// TwinCAT 3 PLC project ccslib
// Title: ESO ELT CCS Library
// Company: ESO
// Author: Mario Kiekebusch
// ProjectVersion: 0.0.1.0
// Description: ELT - CCS Library providing FB helping to receive deterministic data via MUDPI.
// ProgramVersion: 3.1.4022.4
// libraries:
//   ESO ELT Utility Library, * (ESO)
//   ESO LDC Common Library, * (ESO)
//   ESO LDC Timer Library, * (ESO)
//   ESO MUDPI Library, * (ESO)
//   Tc2_EtherCAT, * (Beckhoff Automation GmbH)
//   Tc2_Standard, * (Beckhoff Automation GmbH)
//   Tc2_System, * (Beckhoff Automation GmbH)
//   Tc2_Utilities, * (Beckhoff Automation GmbH)
//   Tc3_Module, * (Beckhoff Automation GmbH)
//   VisuDialogs, * (System)
//   VisuSymbols,3.5.10.0,System
// project tree:
//   DUTs/Structures/ T_CCS_GUI.TcDUT, T_DATA_SAMPLE.TcDUT
//   / GlobalTextList.TcGTLO, VisualizationManager.TcVMO (not stored)
//   GVLs/ GCL.TcGVL, GVL_TimeConstants.TcGVL
//   POUs/ FB_CCS_RECEIVER.TcPOU, FB_LINEAR_INTERPOLATION.TcPOU, MAIN.TcPOU
//   Version/ Global_Version.TcGVL
//   VISUs/Templates/ GUI_TEMPLATE_CCS_RECEIVER.TcVIS

// ---- DUTs/Structures/T_CCS_GUI.TcDUT
TYPE T_CCS_GUI :
STRUCT
	alt: LREAL;
	az: LREAL;
	pa: LREAL;
	time_tai: STRING;
	lst: LREAL;
	ra: LREAL;
	dec: LREAL;
	north_angle: LREAL;
	pupil_angle: LREAL;
	ha: LREAL;
END_STRUCT
END_TYPE

// ---- DUTs/Structures/T_DATA_SAMPLE.TcDUT
TYPE T_DATA_SAMPLE :
STRUCT
	value: LREAL := 0.0;
	timestamp: LREAL := 0.0;
END_STRUCT
END_TYPE

// ---- GVLs/GCL.TcGVL
{attribute 'qualified_only'}
VAR_GLOBAL
	C_PI:				LREAL := 3.1415926535897932384626433832795028841971693993751;
    C_PI2: 				LREAL := C_PI / 2.0;
	C_2PI: 				LREAL := 2.0 * C_PI;
END_VAR

// ---- GVLs/GVL_TimeConstants.TcGVL
{attribute 'qualified_only'}
VAR_GLOBAL
	C_INVALID:    DINT := -9999;
	C_ONE_SEC:    LINT := 1000000000;
	C_STAT_OK:    DINT := 0;
	C_NS2MSEC:    LREAL := 1/1E+6;
	C_NS2SEC:     LREAL := 1/1E+9;
	C_UNIX_OFFSET_SEC: ULINT := DATE_TO_ULINT(DATE#2000-01-01); // 946,684,800 seconds = 15,778,080 minutes = 262,968 hours
	C_UNIX_OFFSET_MICROSEC:  ULINT := C_UNIX_OFFSET_SEC * 10#1000_000;
END_VAR

// ---- Version/Global_Version.TcGVL
{attribute 'TcGenerated'}
{attribute 'no-analysis'}
{attribute 'linkalways'}
// This function has been automatically generated from the project information.
VAR_GLOBAL CONSTANT
	{attribute 'const_non_replaced'}
	stLibVersion_ESO_ELT_CCS_Library : ST_LibVersion := (iMajor := 0, iMinor := 0, iBuild := 1, iRevision := 0, nFlags := 0, sVersion := '0.0.1.0');
END_VAR

// ---- POUs/FB_CCS_RECEIVER.TcPOU
FUNCTION_BLOCK FB_CCS_RECEIVER
VAR_INPUT
	refTimeObj  : REFERENCE TO FB_TIME; 
END_VAR
VAR_OUTPUT
END_VAR
VAR
	fbMudpiReceiver: FB_MUDPI_RECEIVER;
	tracking_raw : T_ASTRO_POINTING_KERNEL_POSITIONS;
	tracking_ccs : T_CCS_GUI;
	north_sample: T_DATA_SAMPLE;
	pupil_sample: T_DATA_SAMPLE;
	pa_sample: T_DATA_SAMPLE;
	north_angle_interpolator: FB_LINEAR_INTERPOLATION;
	pupil_angle_interpolator: FB_LINEAR_INTERPOLATION;
	pa_angle_interpolator: FB_LINEAR_INTERPOLATION;
	previous_sample_id: UDINT := 0;
	
	
  
	
	
END_VAR

// Listen for MUDPI packages
// It assumes data will contain the structure of the CCS ICD
fbMudpiReceiver();

// Get parameters
GetParams();

// Set parameters
SetParams();

METHOD FB_init : BOOL
VAR_INPUT
	bInitRetains : BOOL; // if TRUE, the retain variables are initialized (warm start / cold start)
	bInCopyCode : BOOL;  // if TRUE, the instance afterwards gets moved into the copy code (online change)
END_VAR
previous_sample_id := 0;
END_METHOD

METHOD GetParams
VAR_INPUT
END_VAR
VAR
	north_angle_result : LREAL;
	pupil_angle_result : LREAL;
	pa_angle_result : LREAL;
	diff_time : LREAL;
END_VAR
// Check if a new sample has been received.
// In this case, values from CCS interface shall be copied 
// to the internal structure (structure_raw).

IF (fbMudpiReceiver.packet_info.sampleId <> previous_sample_id) THEN
	memcpy(ADR(tracking_raw), fbMudpiReceiver.GetMudpiPayload(), fbMudpiReceiver.GetMudpiPayloadSize());
	north_sample.value := tracking_raw.north_angle;
	north_sample.timestamp := tracking_raw.time_tai;
	north_angle_interpolator.AddSample(north_sample);

	pupil_sample.value := tracking_raw.pupil_angle;
	pupil_sample.timestamp := tracking_raw.time_tai;
	pupil_angle_interpolator.AddSample(pupil_sample);
	pa_sample.value := tracking_raw.parallactic_angle;
	pa_sample.timestamp := tracking_raw.time_tai;
	pa_angle_interpolator.AddSample(pa_sample);
	
	north_angle_interpolator.Extrapolate(lrTimestamp:=refTimeObj.stat.lrTaiUnixTimeinSecs, lrValue=>north_angle_result);
	pupil_angle_interpolator.Extrapolate(lrTimestamp:=refTimeObj.stat.lrTaiUnixTimeinSecs, lrValue=>pupil_angle_result);
	pa_angle_interpolator.Extrapolate(lrTimestamp:=refTimeObj.stat.lrTaiUnixTimeinSecs, lrValue=>pa_angle_result);
	
	// Interpolating only PA, NORTH and PUPIL angles for the time being. 
	// All the other tracking data are exactly as received.
	tracking_ccs.alt := RAD_TO_DEG(tracking_raw.target_observed_altaz[0]);
	tracking_ccs.az := RAD_TO_DEG(tracking_raw.target_observed_altaz[1]);
	tracking_ccs.pa := RAD_TO_DEG(pa_angle_result);
	tracking_ccs.ra:= F_Rad2Hms(tracking_raw.radec_at_altaz_at_requested_xy[0]);
	tracking_ccs.dec := F_Rad2Dms(tracking_raw.radec_at_altaz_at_requested_xy[1]);
	tracking_ccs.north_angle := RAD_TO_DEG(north_angle_result);
	tracking_ccs.pupil_angle := RAD_TO_DEG(pupil_angle_result);	
	tracking_ccs.time_tai := DCTIME64_TO_STRING(refTimeObj.MudpiTimeToDc(tracking_raw.time_tai));
	tracking_ccs.ha := tracking_raw.time_lst - tracking_raw.radec_at_altaz_at_requested_xy[0];
	previous_sample_id := fbMudpiReceiver.packet_info.sampleId;
	diff_time := tracking_raw.time_tai - refTimeObj.stat.lrTaiUnixTimeinSecs;
ELSE
	north_angle_interpolator.Extrapolate(lrTimestamp:=refTimeObj.stat.lrTaiUnixTimeinSecs, lrValue=>north_angle_result);
	pupil_angle_interpolator.Extrapolate(lrTimestamp:=refTimeObj.stat.lrTaiUnixTimeinSecs, lrValue=>pupil_angle_result);
	pa_angle_interpolator.Extrapolate(lrTimestamp:=refTimeObj.stat.lrTaiUnixTimeinSecs, lrValue=>pa_angle_result);
	
	north_sample.value := north_angle_result;
	north_sample.timestamp := refTimeObj.stat.lrTaiUnixTimeinSecs;
	north_angle_interpolator.AddSample(north_sample);

	pupil_sample.value := pupil_angle_result;
	pupil_sample.timestamp := refTimeObj.stat.lrTaiUnixTimeinSecs;
	pupil_angle_interpolator.AddSample(pupil_sample);
	
	pa_sample.value := pa_angle_result;
	pa_sample.timestamp := refTimeObj.stat.lrTaiUnixTimeinSecs;
	pa_angle_interpolator.AddSample(pa_sample);
	
	tracking_ccs.pa := RAD_TO_DEG(pa_angle_result);
	tracking_ccs.north_angle := RAD_TO_DEG(north_angle_result);
	tracking_ccs.pupil_angle := RAD_TO_DEG(pupil_angle_result);
END_IF
END_METHOD

METHOD SetParams
VAR_INPUT
END_VAR
END_METHOD

END_FUNCTION_BLOCK

// ---- POUs/FB_LINEAR_INTERPOLATION.TcPOU
FUNCTION_BLOCK FB_LINEAR_INTERPOLATION
VAR_INPUT
END_VAR
VAR_OUTPUT
END_VAR
VAR
	x0:	T_DATA_SAMPLE;
	x1: T_DATA_SAMPLE;
	size:  UINT := 0;
END_VAR

METHOD AddSample : BOOL
VAR_INPUT
	sample: T_DATA_SAMPLE;
END_VAR

VAR
	
END_VAR
IF (size = 0) THEN
	x0 := sample;
	size := size + 1;
ELSIF (size = 1) THEN
	x1 := sample;
	size := size + 1;
ELSIF (size = 2) THEN
	x0 := x1;
	x1 := sample;
END_IF
END_METHOD

METHOD Extrapolate 
VAR_INPUT
lrTimestamp: LREAL;
END_VAR
VAR_OUTPUT
    bOk        : BOOL;
    lrValue    : LREAL;
END_VAR
VAR
	tmp        : LREAL;
END_VAR
bOk := FALSE;
IF (size = 0) THEN
	lrValue := 0;
ELSIF (size = 1) THEN
	lrValue := x0.value;
ELSIF (size = 2) THEN
	IF ((x1.timestamp - x0.timestamp) <> 0)  AND ((x1.value - x0.value) <> 0)  THEN
		tmp := x0.value + (lrTimestamp - x0.timestamp) / (x1.timestamp - x0.timestamp) * (x1.value - x0.value);
		lrValue := tmp;
		bOk := TRUE;
	END_IF
END_IF
END_METHOD

METHOD FB_init : BOOL
VAR_INPUT
	bInitRetains : BOOL; // if TRUE, the retain variables are initialized (warm start / cold start)
	bInCopyCode : BOOL;  // if TRUE, the instance afterwards gets moved into the copy code (online change)
END_VAR
VAR
	sample: T_DATA_SAMPLE;
END_VAR
sample.value := 2.7;
sample.timestamp := 1.2;
AddSample(sample);
sample.value := 3.1;
sample.timestamp := 1.4;
AddSample(sample);
sample.value := 2.7;
sample.timestamp := 1.2;
AddSample(sample);
END_METHOD

END_FUNCTION_BLOCK

// ---- POUs/MAIN.TcPOU
PROGRAM MAIN
VAR
	fbMudpiReceiver: FB_MUDPI_RECEIVER;
END_VAR

fbMudpiReceiver();

END_PROGRAM

// ---- GlobalTextList.TcGTLO
TEXTLIST GlobalTextList
  970 = ' Mode:'
  595 = '%.0f'
  599 = '%.1f'
  902 = '%.2e'
  597 = '%.2f'
  508 = '%.3f'
  456 = '%.4f'
  895 = '%.5f'
  510 = '%.6f'
  583 = '%d'
  120 = '%e'
  577 = '%s'
  220 = '.library ver. %s'
  438 = 'Active time: Local'
  645 = 'Active time: Simulated'
  976 = 'Active time: UTC'
  938 = 'Actual'
  441 = 'Address Type'
  681 = 'Admin'
  607 = 'Alt :'
  1042 = 'Ambient'
  956 = 'Angles'
  1009 = 'App Tag'
  2270 = 'Apparent Coordinates'
  1435 = 'Apparent Declination [ddmmss]'
  12 = 'Apparent Declination [rad]'
  207 = 'Apparent Right Ascension [hhmmss]'
  785 = 'Apparent Right Ascension [rad]'
  596 = 'Atmospheric Pressure [mbar]'
  598 = 'Atmospheric Relative Humidity [0..1]'
  601 = 'Atmospheric Temperature [deg C]'
  608 = 'Az :'
  337 = 'CCS library ver. %s'
  824 = 'CCS Simulator'
  746 = 'Component ID'
  1035 = 'Copy current Local time to "New Time"'
  1125 = 'Copy current UTC time to "New Time"'
  652 = 'Copy Local'
  482 = 'Copy UTC'
  1353 = 'Dec :'
  591 = 'Dec:'
  612 = 'Delay Mechanism'
  1119 = 'Dest Port'
  1190 = 'Deterministic Data'
  743 = 'Disable'
  1047 = 'Disable Diagnostics'
  903 = 'Disabled'
  218 = 'DROT Status'
  2033 = 'Dut:'
  587 = 'ELEV'
  586 = 'Elevation Mode:  WHITE=Not Active\nGREEN=Activated'
  536 = 'Enable'
  742 = 'Enable Diagnostics'
  537 = 'Enabled'
  584 = 'ENG'
  579 = 'Engineering Mode:  WHITE=Not active\nGREEN=Activated'
  1794 = 'Equinox'
  520 = 'Equinox:'
  392 = 'Error Message'
  568 = 'Ethernet driver initialization'
  134 = 'Ethernet Settings:'
  381 = 'External Port'
  494 = 'format: '
  57 = 'format: YYYY-MM-DD-hh:mm:ss.nnnnnnnnn'
  311 = 'Frame '
  963 = 'Frame ID '
  66 = 'Gateway'
  594 = 'Humidity :'
  750 = 'Humidity [%]'
  229 = 'Instance name: %s'
  787 = 'Instance: %s'
  505 = 'IP address'
  924 = 'Lapse Rate'
  395 = 'Lapserate:'
  582 = 'Leap Second:'
  407 = 'Local'
  1751 = 'Local Sidereal Time [h]'
  576 = 'Local Time:'
  298 = 'Local:'
  894 = 'LST :'
  531 = 'Mean Coordinates'
  998 = 'Mean Declination [ddmmss]'
  2704 = 'Mean Right Ascension [hhmmss]'
  629 = 'mms'
  578 = 'Mode:'
  935 = 'Motor.library ver. %s'
  644 = 'ms'
  387 = 'MUDPI Receiver'
  552 = 'Net Mask'
  662 = 'New Time'
  854 = 'New Time:'
  625 = 'None'
  103 = 'Nord:'
  261 = 'North angle [deg]'
  104 = 'North angle [rad]'
  164 = 'Not Connected'
  555 = 'Not Synchronized'
  355 = 'Not Syncronized'
  396 = 'Offset from Master'
  551 = 'Offset from Master:'
  71 = 'Operator'
  604 = 'PA :'
  43 = 'Packet Counter'
  703 = 'Packet Info'
  603 = 'Parallactic Angle [deg]'
  205 = 'Parallactic Angle [rad]'
  1057 = 'Payload size'
  231 = 'PLC Port'
  593 = 'Pressure :'
  2321 = 'Pressure [mbar]'
  1012 = 'Pressure:'
  446 = 'PTP Configuration'
  359 = 'PTP Diagnostics'
  467 = 'PTP Version'
  1715 = 'Pupil angle[deg]'
  56 = 'Pupil angle[rad]'
  711 = 'Pupil:'
  2102 = 'Ra :'
  590 = 'Ra:'
  1557 = 'Raw Deterministic Data'
  115 = 'RED - False\nGREEN - True'
  1156 = 'Sample ID'
  893 = 'Sampling'
  876 = 'Service'
  136 = 'Simulation'
  263 = 'Size'
  588 = 'SKY'
  585 = 'Sky Mode:  WHITE=Not Active\nGREEN=Activated'
  589 = 'STAT'
  275 = 'State'
  609 = 'State:'
  580 = 'Stationary Mode:  WHITE=Not Active\nGREEN=Activated'
  81 = 'Stationary Mode:  WHITE=Not Active\nRED=Activated'
  936 = 'Substate:'
  1699 = 'TAI time '
  448 = 'TAI time [sec]'
  331 = 'TAI:'
  937 = 'Target'
  605 = 'TEL Altitude [deg]'
  648 = 'TEL Altitude [rad]'
  606 = 'TEL Azimuth [deg]'
  873 = 'TEL Azimuth [rad]'
  602 = 'TEL Dec'
  600 = 'TEL RA'
  592 = 'Temperature :'
  254 = 'Temperature [degC]'
  1727 = 'Temperature:'
  741 = 'Time'
  664 = 'TIME Mode'
  581 = 'Time Mode:'
  673 = 'TIME Set Mode'
  145 = 'TIME Status'
  800 = 'Time used for Simulation. '
  749 = 'Time used for Simulation. \nPress "Copy UTC" or "Copy Local" button to get the time in correct format and then modify it for your needs.'
  613 = 'timer library ver. %s'
  362 = 'Timer library ver. %s'
  184 = 'Timestamp'
  671 = 'Topic ID'
  945 = 'Tracking mode (=2)'
  442 = 'Transport Layer'
  239 = 'TRS address'
  759 = 'TRS Diagnostics'
  82 = 'TRS Port'
  611 = 'ubstate'
  322 = 'UDP Receiver'
  1124 = 'UDP Sender'
  405 = 'Use local time'
  314 = 'Use simulated time given under "New Time"'
  1002 = 'Use simulated time given under "New Time".\nNOTE: "New Time" is taken only if the time string has been modified since the last press of the button.'
  509 = 'Use UTC time'
  940 = 'USER'
  939 = 'User defined Mode: WHITE=Not Active\nGREEN=Activated'
  983 = 'User Deterministic Data'
  610 = 'UTC'
  691 = 'UTC time [sec]'
  219 = 'UTC:'
  907 = 'Version'
  1720 = 'Wavelength:'
  44 = 'WHITE - Disabled'
  356 = 'WHITE - Disabled\nGREEN - Enabled'
  898 = 'WHITE=Connected\nRED=Not Connected'
  616 = 'WHITE=Synchronized\nRED=Not Synchronized'
  669 = '[ms]'
  950 = '[ns]'
  709 = '[s]'
END_TEXTLIST

// ---- VISUs/Templates/GUI_TEMPLATE_CCS_RECEIVER.TcVIS
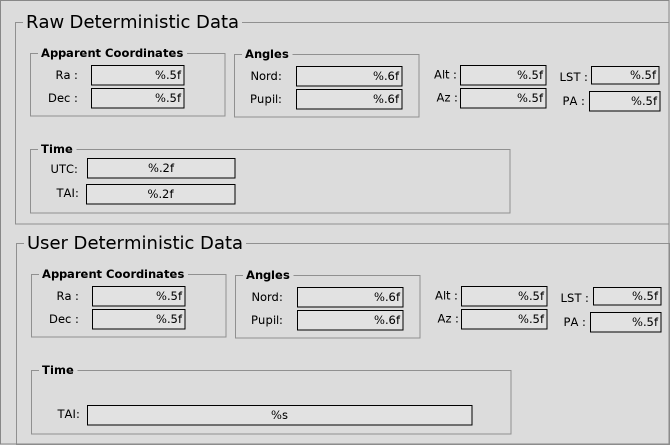
VISUALIZATION GUI_TEMPLATE_CCS_RECEIVER  // 670x445
VAR_INPUT
	m_DeviceName : STRING;
END_VAR
VAR_IN_OUT
	m_Instance : FB_CCS_SIM;
END_VAR
    GroupBox (16,235 654x210), "User Deterministic Data"
        GroupBox (15,31 195x71), "Apparent Coordinates"
            Label (11,20 40x20), "Ra :"
            Label (11,43 40x20), "Dec :"
            Label (8,70 60x20)
            Rectangle (61,43 93x20), "%.5f", tooltip "Apparent Declination [ddmmss]", text variable: m_Instance.tracking_ccs.dec
            Rectangle (61,20 93x20), "%.5f", tooltip "Apparent Right Ascension [hhmmss]", text variable: m_Instance.tracking_ccs.ra
        Rectangle (574,77 71x20), "%.5f", tooltip "Parallactic Angle [deg]", text variable: m_Instance.tracking_ccs.pa
        Label (523,77 50x20), "PA :"
        Label (408,51 37x19), "Alt :"
        Label (411,74 35x19), "Az :"
        Rectangle (445,74 86x20), "%.5f", tooltip "TEL Azimuth [deg]", text variable: m_Instance.tracking_ccs.az
        Rectangle (445,51 86x20), "%.5f", tooltip "TEL Altitude [deg]", text variable: m_Instance.tracking_ccs.alt
        GroupBox (15,127 480x72), "Time"
            Label (6,42 46x20), "TAI:"
            Label (8,70 60x20)
            Rectangle (56,43 385x20), "%s", tooltip "TAI time", text variable: m_Instance.tracking_ccs.time_tai
        GroupBox (219,32 185x71), "Angles"
            Label (11,20 40x20), "Nord:"
            Label (11,43 40x20), "Pupil:"
            Label (8,70 60x20)
            Rectangle (62,20 106x20), "%.6f", tooltip "North angle [deg]", text variable: m_Instance.tracking_ccs.north_angle
            Rectangle (62,43 106x20), "%.6f", tooltip "Pupil angle[deg]", text variable: m_Instance.tracking_ccs.pupil_angle
        Label (534,53 42x20), "LST :"
    GroupBox (15,14 654x210), "Raw Deterministic Data"
        GroupBox (15,31 195x71), "Apparent Coordinates"
            Label (11,20 40x20), "Ra :"
            Label (11,43 40x20), "Dec :"
            Label (8,70 60x20)
            Rectangle (61,43 93x20), "%.5f", tooltip "Apparent Declination [rad]", text variable: m_Instance.tracking_raw.radec_at_altaz_at_requested_xy[1]
            Rectangle (61,20 93x20), "%.5f", tooltip "Apparent Right Ascension [rad]", text variable: m_Instance.tracking_raw.radec_at_altaz_at_requested_xy[0]
        Rectangle (574,77 71x20), "%.5f", tooltip "Parallactic Angle [rad]", text variable: m_Instance.tracking_raw.parallactic_angle
        Label (523,77 50x20), "PA :"
        Label (408,51 37x19), "Alt :"
        Label (411,74 35x19), "Az :"
        Rectangle (445,74 86x20), "%.5f", tooltip "TEL Azimuth [rad]", text variable: m_Instance.tracking_raw.current_observed_altaz[1]
        Rectangle (445,51 86x20), "%.5f", tooltip "TEL Altitude [rad]", text variable: m_Instance.tracking_raw.current_observed_altaz[0]
        GroupBox (15,127 480x72), "Time"
            Label (11,18 40x20), "UTC:"
            Label (6,42 46x20), "TAI:"
            Label (8,70 60x20)
            Rectangle (57,17 148x20), "%.2f", tooltip "UTC time [sec]", text variable: m_Instance.tracking_raw.time_utc
            Rectangle (56,43 149x20), "%.2f", tooltip "TAI time [sec]", text variable: m_Instance.tracking_raw.time_tai
        GroupBox (219,32 185x71), "Angles"
            Label (11,20 40x20), "Nord:"
            Label (11,43 40x20), "Pupil:"
            Label (8,70 60x20)
            Rectangle (62,20 106x20), "%.6f", tooltip "North angle [rad]", text variable: m_Instance.tracking_raw.north_angle
            Rectangle (62,43 106x20), "%.6f", tooltip "Pupil angle[rad]", text variable: m_Instance.tracking_raw.pupil_angle
        Label (534,53 42x20), "LST :"
        Rectangle (578,273 68x18), "%.5f", tooltip "Local Sidereal Time [h]", text variable: m_Instance.tracking_ccs.lst
    Rectangle (591,66 68x18), "%.5f", tooltip "Local Sidereal Time [h]", text variable: m_Instance.tracking_raw.time_lst
END_VISUALIZATION
